FUNCTION_BLOCK POU4
VAR_INPUT
END_VAR
VAR_OUTPUT
END_VAR
VAR
END_VAR

END_FUNCTION_BLOCK

(* stored: Version 1.1.0.1, ProductVersion 3.1.4020.12
   POU POU4: Id {2e7b3a82-d1bb-4ef3-bb60-e7bf52f565b7}, SpecialFunc None *)
